(* PLC project Main, Beckhoff Automation GmbH TwinCAT PLC Control 3.5.13.21 *)
(* stored: creationDateTime 2022-06-12T18:07:28.7209284, modificationDateTime 2022-06-12T18:07:28.7229285 *)

PROGRAM MAIN
VAR
	velocity		AT%I*	: INT;		// nDataOut2[0] . nDataOut2 . Out . Ausgänge . Drive . ConveyorMotorAxis . ConveyorMotorAxis . Achsen . NC-Task 1 SAF
	counterValue 	AT%Q*	: UINT := 0;		//nDataIn1[0] . nDataIn1 . In . Eingänge . Enc . ConveyorMotorAxis . ConveyorMotorAxis . Achsen . NC-Task 1 SAF
	driveInState1	AT%Q*	: USINT;	// State of the hardware motor module
	
	
	ModelToPLC		: DWORD := 0;		// empty (1), driveInState1 (1), counterValue (2)
	PLCToModel		: DWORD := 0;		// empty (2), velocity (2)
END_VAR

            // Communication
// ToPlc
counterValue := DWORD_TO_UINT(ModelToPLC AND 16#00_00_FF_FF);
driveInState1 := DWORD_TO_USINT(SHR((ModelToPLC AND 16#00_FF_00_00),16));


// ToModel
PLCToModel := 0;
PLCToModel := SHL((PLCToModel OR velocity),0);
          
END_PROGRAM
